FUNCTION_BLOCK ARRAY2VALUES_2_LREAL (* Service Interface Function Block Type *)
  (* Standard: 61499-2 *)
  (* Version 0.0, 2014-06-13, 4DIAC-IDE, 4DIAC-Consortium *)
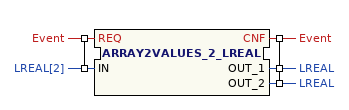
  EVENT_INPUT
    REQ WITH IN; (* Service Request *)
  END_EVENT
  EVENT_OUTPUT
    CNF WITH OUT_1, OUT_2; (* Confirmation of Requested Service *)
  END_EVENT
  VAR_INPUT
    IN : ARRAY [0..1] OF LREAL; (* Array input *)
  END_VAR
  VAR_OUTPUT
    OUT_1 : LREAL; (* output number 1 *)
    OUT_2 : LREAL; (* output number 2 *)
  END_VAR
  (* Service APPLICATION/RESOURCE: Service Interface Function Block Type *)
END_FUNCTION_BLOCK
